INTERFACE I_OPCUA_NodeGetHandle

METHOD start : BOOL
VAR_INPUT
    Execute       : BOOL;
    ConnectionHdl : DWORD;
    NodeID        : ST_UANodeID;
    Timeout       : TIME := DEFAULT_ADS_TIMEOUT; 
END_VAR 
VAR_OUTPUT
    NodeHdl     : DWORD;
    Done        : BOOL;
    Busy        : BOOL;
    Error       : BOOL;
    ErrorID     : DWORD;
END_VAR
END_METHOD

END_INTERFACE

(* stored: Version 1.1.0.1, ProductVersion 3.1.4024.9
   Itf I_OPCUA_NodeGetHandle: Id {3d2ebc4d-3aa1-4e39-9753-516fea065d45}
   Method start: Id {031056aa-9ef3-4a25-8b9a-d2f2930a2b4c} *)
